Staubli VAL3: sendAck.pgx

public program sendAck(num& x_nMsgRecvState)
begin
  // Copyright (c) 2016, Ocado Technology - Robotics Research Team
  //
  // Licensed under the Apache License, Version 2.0 (the "License");
  // you may not use this file except in compliance with the License.
  // You may obtain a copy of the License at
  //
  //     http://www.apache.org/licenses/LICENSE-2.0
  //
  // Unless required by applicable law or agreed to in writing, software
  // distributed under the License is distributed on an "AS IS" BASIS,
  // WITHOUT WARRANTIES OR CONDITIONS OF ANY KIND, either express or implied.
  // See the License for the specific language governing permissions and
  // limitations under the License.



  switch rosGenericMsg.header.nMsgType
    case nStdMsgType["JOINT_TRAJ_PT"]
      call sendRosMsg(siTcpIpMotion,rosTrajPtAck.prefix,rosTrajPtAck.header,rosTrajPtAck.body,nInConnFlag)
    break
    case nStdMsgType["JOINT_TRAJ_PT_FULL"]
      call sendRosMsg(siTcpIpMotion,rosTrajPtFAck.prefix,rosTrajPtFAck.header,rosTrajPtFAck.body,nInConnFlag)
    break
    default
    break
  endSwitch

  // regardless of result from sending ACK
  // reset state machine to receive new messages
  x_nMsgRecvState=nReset
end
